{attribute 'enable_dynamic_creation'}
FUNCTION_BLOCK FB_TaskMoveZ EXTENDS FB_AbstructFuture
VAR_OUTPUT
END_VAR
VAR
	_v				: MC_LREAL;
	_a				: MC_LREAL;
	_d				: MC_LREAL;
	_j				: MC_LREAL;
	_dynamics		: DynamicConstraint_PathXY;
	_position 		: LREAL;
	_error_id		: UDINT;
	_mover			: REFERENCE TO MC_PlanarMover;
	_cmdFB			: MC_PlanarFeedback;
	_prohibit 		: BOOL;
	_abort_executor : FB_Executor;
	_state_num 			:UINT;
	_abort_state	:UINT;
END_VAR

{warning 'add method implementation '}
METHOD abort : BOOL
_cmdFB.Update();
_state_num := 0;
CASE _abort_state OF
	0:
		IF _cmdFB.Active THEN
			_dynamics.SetValuesVADJ(2000,20000,200000,200000);
			_abort_state := 1;
		ELSE
			abort := TRUE;
		END_IF
	1:
		//停止
		_mover.Halt(_cmdFB,_dynamics);
		_abort_state := 2;
	2:
		//停止完了フラグ待ち
		IF _cmdFB.Done THEN
			abort := TRUE;
			_error_id := 0;
		END_IF
		IF _cmdFB.Error THEN
			abort := TRUE;
			_error_id := _cmdFB.ErrorId;
		END_IF
END_CASE
END_METHOD

{warning 'add method implementation '}
METHOD execute : BOOL
_cmdFB.Update();
_abort_state := 0;
CASE _state_num OF
	0:
		//直線運動
		IF NOT _cmdFB.Active AND NOT _cmdFB.Busy THEN
			_mover.MoveZ(_cmdFB,_position,_dynamics);
			_state_num := 1;
		END_IF
	1:
		//直線運動の完了フラグ待ち
		IF _cmdFB.Done THEN
			execute := TRUE;
			_error_id := 0;
		END_IF
		IF _cmdFB.Error THEN
			execute := TRUE;
			_error_id := _cmdFB.ErrorId;
		END_IF
END_CASE
END_METHOD

{warning 'add method implementation '}
METHOD init : BOOL
IF _prohibit THEN
	_error_id := 16#80000000;
	init := TRUE;
ELSIF _v = 0 OR _a = 0 OR _d = 0 THEN
	_error_id := 1;
	init := TRUE;
ELSE
	_dynamics.SetValuesVADJ(_v, _a, _d, _j);
	_abort_executor.init();
	_error_id := 0;
	_state_num := 0;
	_abort_state := 0;
	init := TRUE;
END_IF
END_METHOD

PROPERTY mover : REFERENCE TO MC_PlanarMover
SET
_mover REF= mover;
END_SET
END_PROPERTY

{warning 'add property implementation'}
PROPERTY nErrorID : UDINT
GET
nErrorID := _error_id;
END_GET
END_PROPERTY

{warning 'add method implementation '}
METHOD quit : BOOL
init();
quit := TRUE;
END_METHOD

METHOD set_dynamics : BOOL
VAR_INPUT
	v: MC_LREAL;
	a: MC_LREAL;
	d: MC_LREAL;
	j: MC_LREAL;
END_VAR
_v := v;
_a := a;
_d := d;
_j := j;
set_dynamics := TRUE;
END_METHOD

METHOD set_target_position : BOOL
VAR_INPUT
	z: LREAL;
END_VAR
_position := z;

set_target_position := TRUE;
END_METHOD

END_FUNCTION_BLOCK

(* stored: Version 1.1.0.1, ProductVersion 3.1.4024.12
   POU FB_TaskMoveZ: Id {12a459c4-2269-493f-a10a-5eeb49730032}, SpecialFunc None
   Method abort: Id {e445749c-5cde-40f7-b4d0-b3be9d689d2f}
   Method execute: Id {0a077d8f-f72d-4e4d-beb6-15d2a4b64571}
   Method init: Id {24dd061e-2fea-44b1-aea3-558e14376613}
   Property mover: Id {c8ab674a-b42c-45f6-93c1-7d0697eb4078}
   Set Set: Id {398ca2ea-4327-414b-83d2-12879ed08847}
   Property nErrorID: Id {707247e6-3bf8-4890-a7bd-3a94a8e3e541}
   Get Get: Id {646bb9ed-52d7-4992-837a-61e732dba46f}
   Method quit: Id {87a32588-77e1-496e-8dea-6434b422710e}
   Method set_dynamics: Id {62a8f046-ff21-4711-b276-c938a914c217}
   Method set_target_position: Id {1eaddfbd-0cdd-4b0f-8f02-fccb562753a5} *)
